FUNCTION_BLOCK SHARED_SWITCH (* Composite Function Block Type *)
  (* Standard: 61499-2 *)
  (* Version 0.0, 2/8/2023, brink, Flexbridge AB, template *)
  PACKAGE UAO.Hackathon;
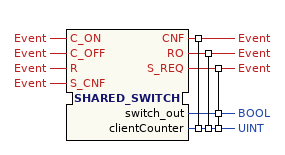
  EVENT_INPUT
    C_ON; (* Increment 'on' counter *)
    C_OFF; (* Decrement 'on' counter *)
    R;
    S_CNF;
  END_EVENT
  EVENT_OUTPUT
    CNF WITH clientCounter; (* Execution Confirmation *)
    RO WITH clientCounter;
    S_REQ WITH switch_out, clientCounter;
  END_EVENT
  VAR_OUTPUT
    switch_out : BOOL; (* Output event qualifier *)
    clientCounter : UINT;
  END_VAR
  FBS
    counter : E_UCNTR(PVL := 0, PVH := 1);
    expect_on_off : E_SWITCH;
    switch_already_on : E_SWITCH;
    switch_already_off : E_SWITCH;
    switch_is_on : E_RS;
    merge_already_correct : E_MERGE;
    merge_set_or_correct : E_MERGE;
    when_switch_set : E_PERMIT;
    switch_setting_or_set : E_SWITCH;
    setting_switch : E_RS;
    switch_is_off : NOT_42C76073DCEB1A7A; {SET_ATTRIBUTE(Configuration.GenericFBType.InterfaceParams, Runtime.Standard#CNT:=1;OUT${CNT$}:BOOL)}
  END_FBS
  EVENT_CONNECTIONS
    C_ON TO counter.CU;
    C_OFF TO counter.CD;
    counter.CUO TO expect_on_off.EI;
    switch_already_off.EO1 TO merge_already_correct.EI1;
    switch_already_on.EO1 TO merge_already_correct.EI2;
    S_CNF TO when_switch_set.EI;
    switch_already_off.EO0 TO switch_is_on.R;
    switch_already_on.EO0 TO switch_is_on.S;
    switch_setting_or_set.EO1 TO S_REQ;
    merge_already_correct.EO TO merge_set_or_correct.EI2;
    switch_setting_or_set.EO0 TO merge_set_or_correct.EI1;
    merge_set_or_correct.EO TO CNF;
    setting_switch.EO TO switch_setting_or_set.EI;
    when_switch_set.EO TO setting_switch.R;
    switch_is_on.EO TO setting_switch.S;
    R TO counter.R;
    counter.RO TO RO;
    expect_on_off.EO1 TO switch_already_on.EI;
    switch_is_off.CNF TO switch_already_off.EI;
    expect_on_off.EO0 TO switch_is_off.REQ;
    counter.CDO TO expect_on_off.EI;
  END_CONNECTIONS
  DATA_CONNECTIONS
    counter.QH TO expect_on_off.G;
    switch_is_on.Q TO switch_out;
    setting_switch.Q TO when_switch_set.PERMIT;
    setting_switch.Q TO switch_setting_or_set.G;
    switch_is_off.OUT1 TO switch_already_off.G;
    switch_is_on.Q TO switch_is_off.IN1;
    switch_is_on.Q TO switch_already_on.G;
    counter.CV TO clientCounter;
  END_CONNECTIONS
END_FUNCTION_BLOCK
